(* PLC project Generated.project, CODESYS CODESYS V3.5 SP19 Patch 1 *)
(* stored: creationDateTime 2026-09-06T13:00:42.523976, modificationDateTime 2026-09-06T13:00:42.523976 *)

(* ═══════════════════════════════════════════════════════════════ 🚦 ST_ModesState — États et diagnostics IHM des modes de marche ═══════════════════════════════════════════════════════════════ *)
TYPE ST_ModesState : STRUCT
  CurrentMode : E_Mode;  (* 🎚️ Mode de marche actuellement actif *)
  AnyFaultActive : BOOL;  (* : au moins un défaut/alarme actif dans le domaine *)
  ModeChangePendingBlocked : BOOL;  (* 🚦 Changement de mode refusé : treuils non à l'arrêt confirmé (contacteurs retombés + frein serré + |v| < seuil) *)
  ModeChangeBlockReason : STRING(40);  (* 🚦 Motif du blocage de bascule (texte court, ex. "Chgt mode refuse : contacteur M1") *)
  M1ContactorsReleased : BOOL;  (* Détail des 6 sous-conditions de ModeChangeAllowed (diagnostic IHM) — TRUE = condition satisfaite M1 : contacteurs retombés *)
  M1BrakeApplied : BOOL;  (* M1 : frein serré *)
  M1SpeedLow : BOOL;  (* M1 : vitesse sous seuil *)
  M2ContactorsReleased : BOOL;  (* M2 : contacteurs retombés *)
  M2BrakeApplied : BOOL;  (* M2 : frein serré *)
  M2SpeedLow : BOOL;  (* M2 : vitesse sous seuil *)
  HomingRequiredM1 : BOOL;  (* 🧭 M1 : re-homing obligatoire avant retour SEMI_AUTO *)
  HomingRequiredM2 : BOOL;  (* 🧭 M2 : re-homing obligatoire avant retour SEMI_AUTO *)
END_STRUCT;
END_TYPE

(* values of E_Mode: DISABLE: Mode Désactivé / Veille de sécurité (sorties bloquées); MAINT_N1: Manuel Niveau 1 : Pilotage unitaire avec toutes sécurités actives; MAINT_N2: Manuel Niveau 2 : Pilotage dégradé (droits étendus + bypasses autorisés); SEMI_AUTO: Mode Semi-Automatique (séquenceur automatique) *)

{attribute 'qualified_only'}
{attribute 'strict'}
TYPE E_Mode : (DISABLE := 0, MAINT_N1 := 1, MAINT_N2 := 2, SEMI_AUTO := 3);
END_TYPE
